(* Logix 5000 project; controller Lab05_anb5567_msw5288 vendor 1 type 14 code 77 rev 20.12; software revision 20.01 *)

TASK MainTask (continuous, watchdog 500 ms) : MainProgram

MODULES
   Controller : vendor 1 type 14 code 77 (CompactLogixL32EController 0, rev 20.12)
      LocalENB : 1769-L32E Ethernet Port (CompactLogixL32Ethernet 1, rev 20.11)
      Local : CompactBus (CompactVirtualAdapter 3, rev 20.11)
         DC_DI_16 : 1769-IQ16 (Compact 2, rev 1.1, Input RPI 20 ms)
         Analog_4I_2O : vendor 1 type 10 code 43 (Compact 1, rev 1.1, Output RPI 80 ms)
         Relay_DO_16 : 1769-OW16 (Compact 3, rev 1.1, Output RPI 20 ms)
         Analog_8Channel : 1769-IF8 (Compact 6, rev 1.1, Output RPI 80 ms)
         IT6C_TAI : vendor 1 type 10 code 36 (Compact 4, rev 1.1, Input RPI 80 ms)   // Thermocouple Input Module
END_MODULES

VAR_GLOBAL   (* controller tags *)
   ALM : DINT;   // Alarms
        .2   // P100 Run Fault
        .1   // Tank 100 high-high level alarm
        .0   // Low Low Level Alarm
   BV100 : BOOL;   // Tank 100 outlet valve(pneumatic solenoid)
   CV101 : BOOL;   // Tank 100 water inlet valve (pnematic solenoid)
   FCV101 : REAL;   // Tank 100 water in heater steam control valve (I/P)
   FT100 : REAL := -0.12483891;   // Tank 100 discharge flow rate (4-20 mA, 0 to 100 gpm)
   FT101 : REAL := -0.18725838;   // Tank 100 water in flow rate (4-20 mA, 0 to 150 gpm)
   gBit : DINT := 2;   // General Purpose Bits
        .2   // P100 IN AUTO
        .3   // Pump Transfer Started
        .4   // Stop (0 = stopped, 1 = OK)
        .5   // System Auto mode
        .0   // Start the Transfer
        .1   // Stop the Transfer
   gTmr : TIMER[10] := ([0].PRE := 3000, [1].PRE := 5000, [2].PRE := 3000, [3].PRE := 2000, [4].PRE := 500, [5].PRE := 500);   // Timers
        [1].DN   // Low Low Alarm Timer
   HMI_HOA_IA : DINT;   // In Auto
        .0   // Inlet Vave In Auto
        .1   // Outlet Valve In Auto
        .2   // Pump In Auto
   HMI_HOA_IH : DINT;   // In Hand
        .0   // Inlet Valve In Hand
        .1   // Outlet Valve In Hand
        .2   // Pump In Hand
   HMI_HOA_IO : DINT;   // In Off
        .0   // Inlet In Off
        .2   // Pump Off
        .1   // Outlet Valve In Off
   HMI_HOA_RA : DINT;   // Request Auto
        .0   // Request Inlet In Auto
        .1   // Request Outlet In Auto
        .2   // Request Pump In Auto
   HMI_HOA_RH : DINT;   // Request Hand
        .0   // Request Inlet In Hand
        .1   // Request Outlet In Hand
        .2   // Request Pump In hand
   HMI_HOA_RO : DINT;   // Request Off
        .0   // Request Inlet In Off
        .1   // Request Outlet OFF
        .2   // Request Pump Off
   HMI_MR : DINT := 2;   // Misc Request
        .0   // Request Transfer Start
        .1   // Request Transfer Stop
        .2   // Request System Auto
        .3   // Request Alarm Acknowledge
   HMI_MS : DINT := 2;   // Misc Status
        .0   // Start Transfer Status
        .1   // Stop Transfer Status
        .2   // System Auto Status
   HMI_PB : DINT;   // HMI Push Buttons
        .0   // CV101 Hand HMI PB
        .1   // CV101 OFF hmi PB
        .2   // CV101 Auto HMI PB
        .3   // BV100 Hand PB
        .4   // BV100 Off PB
        .5   // BV100 In Auto PB
        .6   // P100 Hand PB
        .7   // P100 OFF PB
        .8   // P100 Auto HMI PB
        .11   // Acknowledge
        .10   // Stop HMI Push Button
        .9   // Transfer HMI Push Button
   HOA_AC : DINT;   // Auto Command
        .0   // Inlet Auto Command
        .1   // Outlet Valve Auto Command
   LSH100 : BOOL;   // Tank 100 high level switch (1= water at switch)
   LSHH100 : BOOL := 1;   // Tank 100 high-high level switch (1= no water at switch)
   LSL100 : BOOL;   // Tank 100 low level switch (1 = water at switch)
   LSLL100 : BOOL := 1;   // Tank 100 low-low level switch (1 = water at switch)
   LT100 : REAL := 6.5884533;   // Tank 100 level (4-20 mA, 0 to 3 psi, 0 to 100% full at 6 ft.w.c.)
   N_ALM : DINT;   // New Alarms
        .2   // New P100 Run Fault
        .0   // New Low Low Level Alarm
        .1   // New Tank 100 high-high level alarm
   P100 : BOOL;   // Tank 100 outlet pump RUN (Motor starter coil)
   P100RNG : BOOL;   // Tank 100 Outlet pump RUNNING (motor starter auxiliary contact)
   PB100A : BOOL;   // Start PB (1 = pressed)
   PB100B : BOOL := 1;   // Stop PB (0 = pressed)
   PL100G : BOOL;   // Green Pilot light
   PL100R : BOOL;   // Red pilot light
   SimConfig : DINT[100];   // Simulation Configuration Data
        [1].0   // SIMULATION 1 = No 480 VAC to MCC
        [1].1   // SIMULATION 1 = Tank 100 disconnect is open
        [1].10   // SIMULATION 1 = LSLL100 switch bad
        [1].11   // SIMULATION 1 = LSL100 switch bad
        [1].12   // SIMULATION 1 = LSH100 switch bad
        [1].13   // SIMULATION 1 = LSHH100 switch bad
        [1].2   // SIMULATION 1 = Tank 100 fuses blown
        [1].3   // SIMULATION 1 = CV101 solenoid valve bad
        [1].4   // SIMULATION 1 = No plant air pressure for control valves
        [1].5   // SIMULATION 1 = BV100 solenoid valve bad
        [1].6   // SIMULATION 1 = Local:3:O 1769-OW16 output card fuse blown
        [1].7   // SIMULATION 1 = PL100G bulb bad
        [1].8   // SIMULATION 1 = PL100R bulb bad
        [1].9   // SIMULATION 1 = Local:2:I 1769-IQ16 +24 VDC to inputs fuse blown
   SimLocal_2_I_Data : INT := 1174;   // SIMULATED INPUTS 1769-IQ16 Local:2:I
        .0   // SIMULATED INPUT Local:2:I.Data.0 Start PB 1 = pressed PB100A
        .1   // SIMULATED INPUT Local:2:I.Data.1 Stop PB 0 = pressed PB100B
        .10   // SIMULATED INPUT Local:2:I.Data.10 Bin 100 outlet slide gate IS CLOSED
        .11   // SIMULATED INPUT Local:2:I.Data.11 Tank 100 agitator RUNNING
        .12   // SIMULATED INPUT Local:2:I.Data.12 spare
        .13   // SIMULATED INPUT Local:2:I.Data.13 spare
        .14   // SIMULATED INPUT Local:2:I.Data.14 spare
        .15   // SIMULATED INPUT Local:2:I.Data.15 spare
        .2   // SIMULATED INPUT Local:2:I.Data.2 Enable SS 1 = Enable SS100
        .3   // SIMULATED INPUT Local:2:I.Data.3 Tank 100 outlet pump RUNNING P100RNG
        .4   // SIMULATED INPUT Local:2:I.Data.4 Tank 100 low-low level switch 1=water at switch LSLL100
        .5   // SIMULATED INPUT Local:2:I.Data.5 Tank 100 low level switch 1=water at switch LSL100
        .6   // SIMULATED INPUT Local:2:I.Data.6 Tank 100 high level switch 1=water at switch LSH100
        .7   // SIMULATED INPUT Local:2:I.Data.7 Tank 100 high-high level switch 1=no water at switch LSHH100
        .8   // SIMULATED INPUT Local:2:I.Data.8 Bin 100 screw conveyor RUNNING
        .9   // SIMULATED INPUT Local:2:I.Data.9 Bin 100 outlet slide gate IS OPEN
   SPD100 : REAL;   // Tank 100 outlet pump speed command (VFD SPEED reference input)
   SS100 : BOOL := 1;   // Enable SS (1=enabled)
   TT100 : REAL := 57.889015;   // Tank 100 product temperature (4-20 mA, 0 to 250 °F)
   TT101 : REAL := 55.986225;   // Tank 100 water in temperature (4-20 mA, 0 to 250 °F)
   TT900 : REAL := 72.518555;   // Room temperature (Type T thermocouple)
   WT100 : REAL := 155.84729;   // Tank 100 weight (4-20 mA, 0 to 10000 lb)
END_VAR

PROGRAM MainProgram   (* main routine MainRoutine *)

ROUTINE AlarmLogic   (* ladder *)
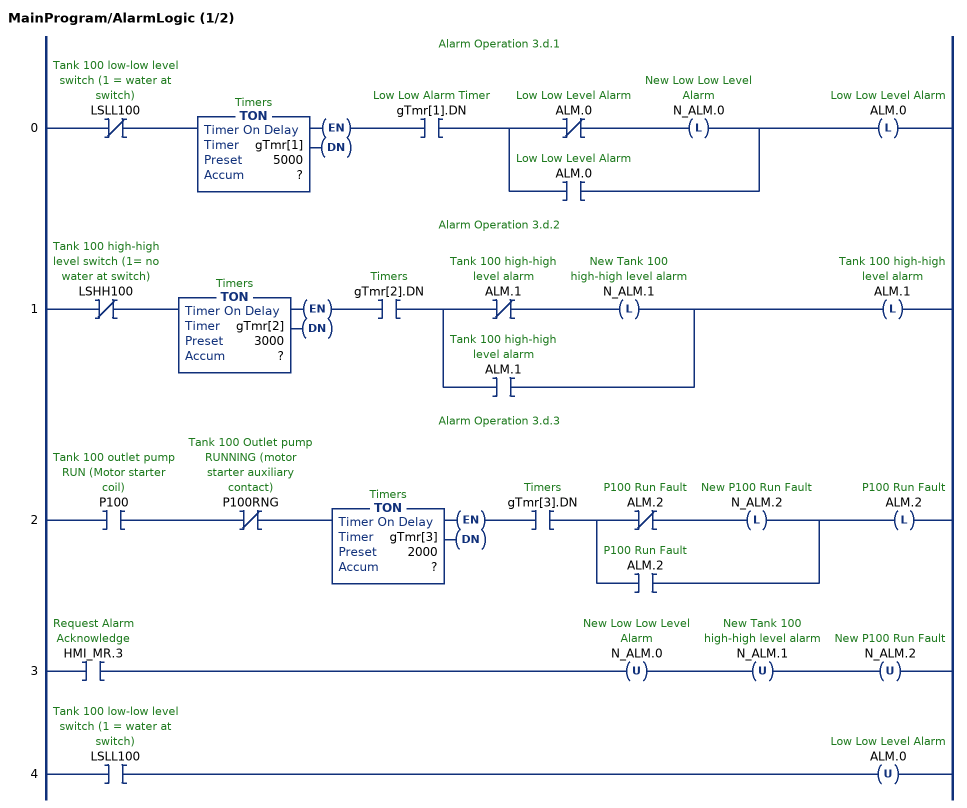
   // Alarm Operation 3.d.1
   0: XIO(LSLL100)TON(gTmr[1],?,?)XIC(gTmr[1].DN)[XIO(ALM.0) OTL(N_ALM.0) ,XIC(ALM.0) ]OTL(ALM.0);
   // Alarm Operation 3.d.2
   1: XIO(LSHH100)TON(gTmr[2],?,?)XIC(gTmr[2].DN)[XIO(ALM.1) OTL(N_ALM.1) ,XIC(ALM.1) ]OTL(ALM.1);
   // Alarm Operation 3.d.3
   2: XIC(P100)XIO(P100RNG)TON(gTmr[3],?,?)XIC(gTmr[3].DN)[XIO(ALM.2) OTL(N_ALM.2) ,XIC(ALM.2) ]OTL(ALM.2);
   3: XIC(HMI_MR.3)OTU(N_ALM.0)OTU(N_ALM.1)OTU(N_ALM.2);
   4: XIC(LSLL100)OTU(ALM.0);
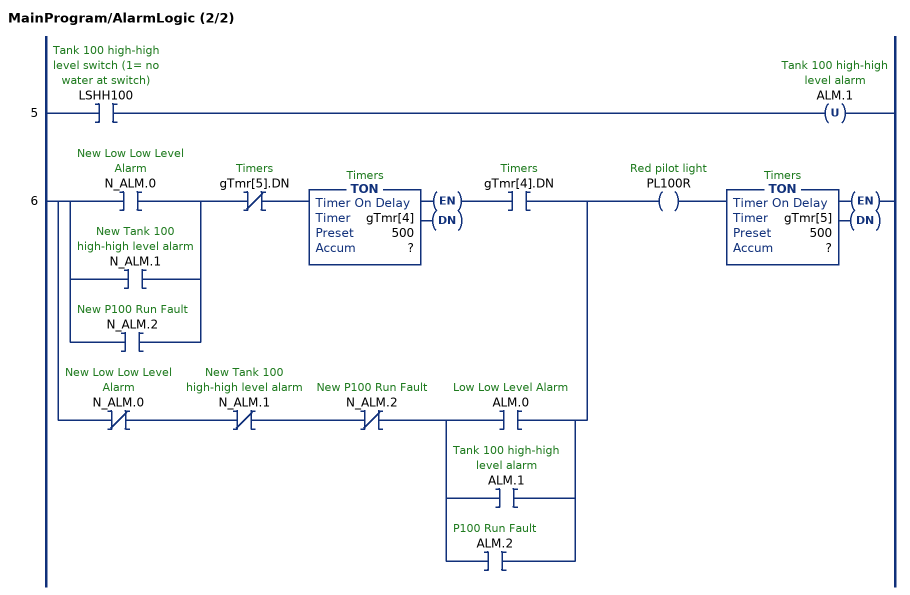
   5: XIC(LSHH100)OTU(ALM.1);
   6: [[XIC(N_ALM.0) ,XIC(N_ALM.1) ,XIC(N_ALM.2) ] XIO(gTmr[5].DN) TON(gTmr[4],?,?) XIC(gTmr[4].DN) ,XIO(N_ALM.0) XIO(N_ALM.1) XIO(N_ALM.2) [XIC(ALM.0) ,XIC(ALM.1) ,XIC(ALM.2) ] ]OTE(PL100R)TON(gTmr[5],?,?);
END_ROUTINE

ROUTINE HMIInputs   (* ladder *)
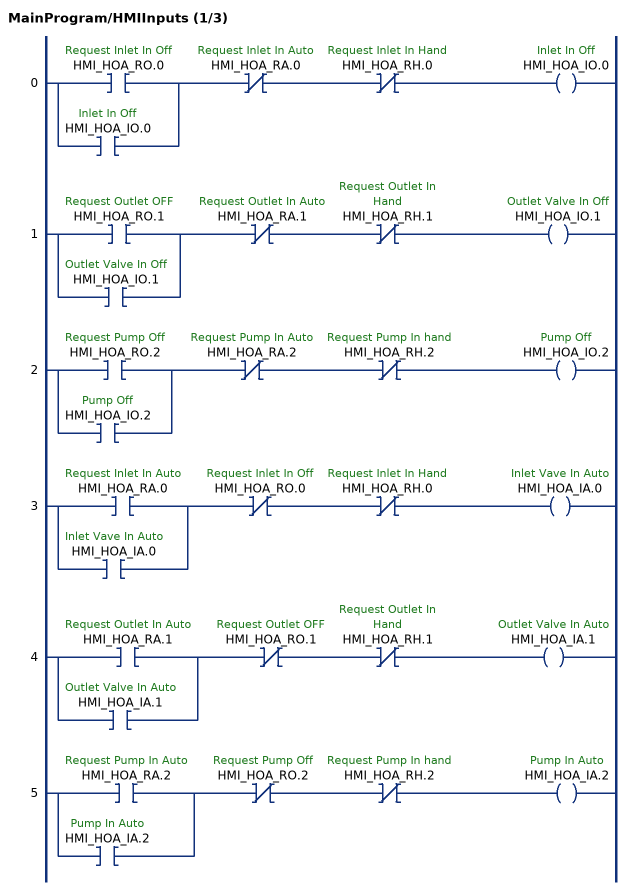
   0: [XIC(HMI_HOA_RO.0) ,XIC(HMI_HOA_IO.0) ]XIO(HMI_HOA_RA.0)XIO(HMI_HOA_RH.0)OTE(HMI_HOA_IO.0);
   1: [XIC(HMI_HOA_RO.1) ,XIC(HMI_HOA_IO.1) ]XIO(HMI_HOA_RA.1)XIO(HMI_HOA_RH.1)OTE(HMI_HOA_IO.1);
   2: [XIC(HMI_HOA_RO.2) ,XIC(HMI_HOA_IO.2) ]XIO(HMI_HOA_RA.2)XIO(HMI_HOA_RH.2)OTE(HMI_HOA_IO.2);
   3: [XIC(HMI_HOA_RA.0) ,XIC(HMI_HOA_IA.0) ]XIO(HMI_HOA_RO.0)XIO(HMI_HOA_RH.0)OTE(HMI_HOA_IA.0);
   4: [XIC(HMI_HOA_RA.1) ,XIC(HMI_HOA_IA.1) ]XIO(HMI_HOA_RO.1)XIO(HMI_HOA_RH.1)OTE(HMI_HOA_IA.1);
   5: [XIC(HMI_HOA_RA.2) ,XIC(HMI_HOA_IA.2) ]XIO(HMI_HOA_RO.2)XIO(HMI_HOA_RH.2)OTE(HMI_HOA_IA.2);
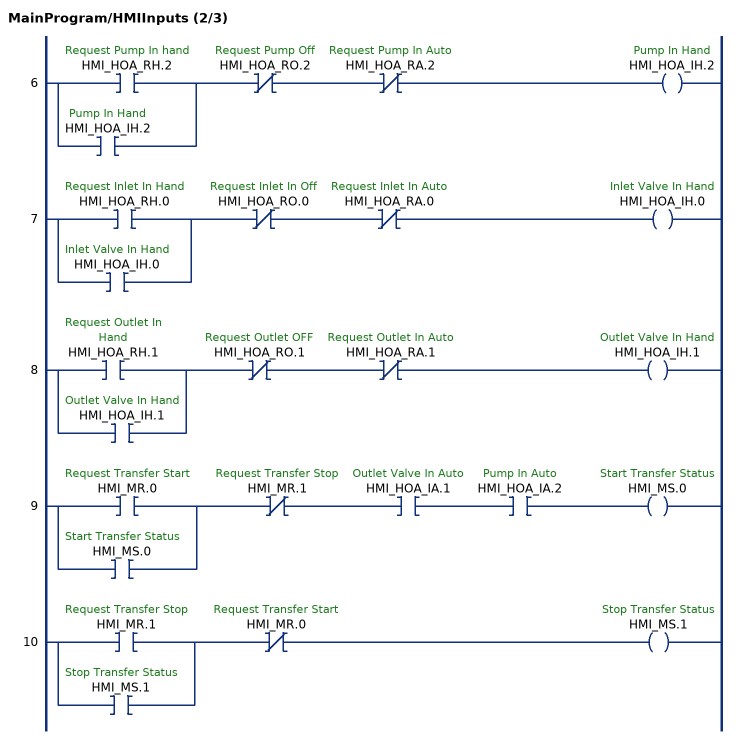
   6: [XIC(HMI_HOA_RH.2) ,XIC(HMI_HOA_IH.2) ]XIO(HMI_HOA_RO.2)XIO(HMI_HOA_RA.2)OTE(HMI_HOA_IH.2);
   7: [XIC(HMI_HOA_RH.0) ,XIC(HMI_HOA_IH.0) ]XIO(HMI_HOA_RO.0)XIO(HMI_HOA_RA.0)OTE(HMI_HOA_IH.0);
   8: [XIC(HMI_HOA_RH.1) ,XIC(HMI_HOA_IH.1) ]XIO(HMI_HOA_RO.1)XIO(HMI_HOA_RA.1)OTE(HMI_HOA_IH.1);
   9: [XIC(HMI_MR.0) ,XIC(HMI_MS.0) ]XIO(HMI_MR.1)XIC(HMI_HOA_IA.1)XIC(HMI_HOA_IA.2)OTE(HMI_MS.0);
   10: [XIC(HMI_MR.1) ,XIC(HMI_MS.1) ]XIO(HMI_MR.0)OTE(HMI_MS.1);
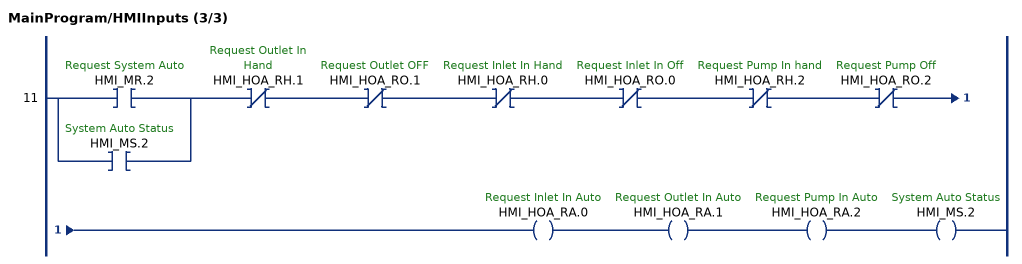
   11: [XIC(HMI_MR.2) ,XIC(HMI_MS.2) ]XIO(HMI_HOA_RH.1)XIO(HMI_HOA_RO.1)XIO(HMI_HOA_RH.0)XIO(HMI_HOA_RO.0)XIO(HMI_HOA_RH.2)XIO(HMI_HOA_RO.2)OTE(HMI_HOA_RA.0)OTE(HMI_HOA_RA.1)OTE(HMI_HOA_RA.2)OTE(HMI_MS.2);
END_ROUTINE

ROUTINE MainRoutine   (* ladder *)
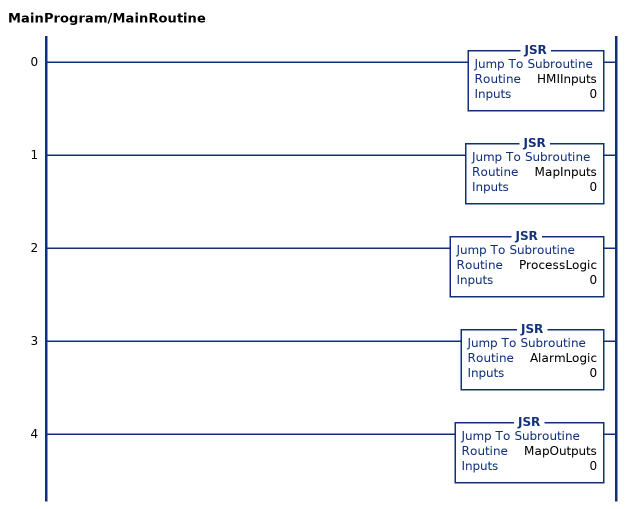
   0: JSR(HMIInputs,0);
   1: JSR(MapInputs,0);
   2: JSR(ProcessLogic,0);
   3: JSR(AlarmLogic,0);
   4: JSR(MapOutputs,0);
END_ROUTINE

ROUTINE MapInputs   (* ladder *)
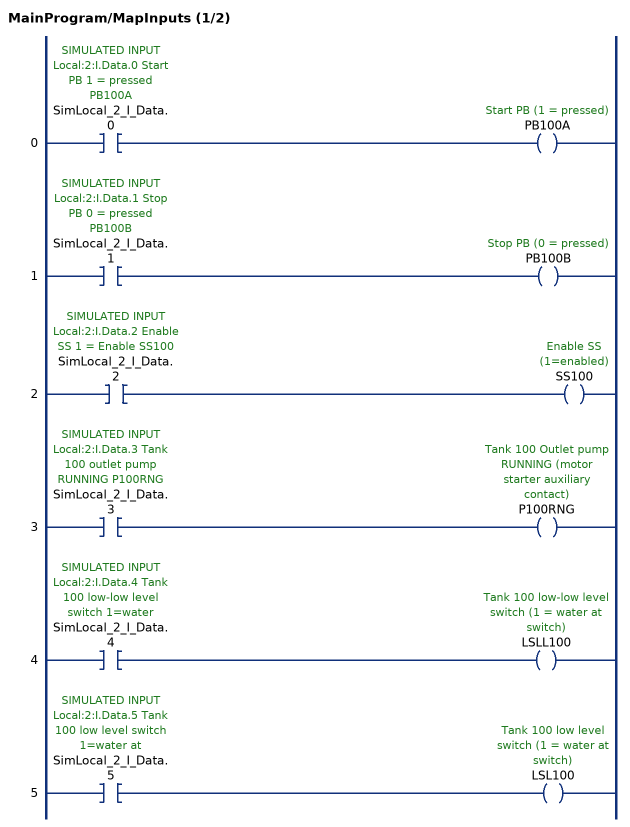
   0: XIC(SimLocal_2_I_Data.0)OTE(PB100A);
   1: XIC(SimLocal_2_I_Data.1)OTE(PB100B);
   2: XIC(SimLocal_2_I_Data.2)OTE(SS100);
   3: XIC(SimLocal_2_I_Data.3)OTE(P100RNG);
   4: XIC(SimLocal_2_I_Data.4)OTE(LSLL100);
   5: XIC(SimLocal_2_I_Data.5)OTE(LSL100);
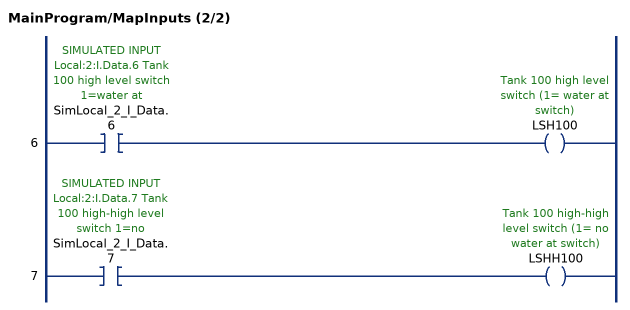
   6: XIC(SimLocal_2_I_Data.6)OTE(LSH100);
   7: XIC(SimLocal_2_I_Data.7)OTE(LSHH100);
END_ROUTINE

ROUTINE MapOutputs   (* ladder *)
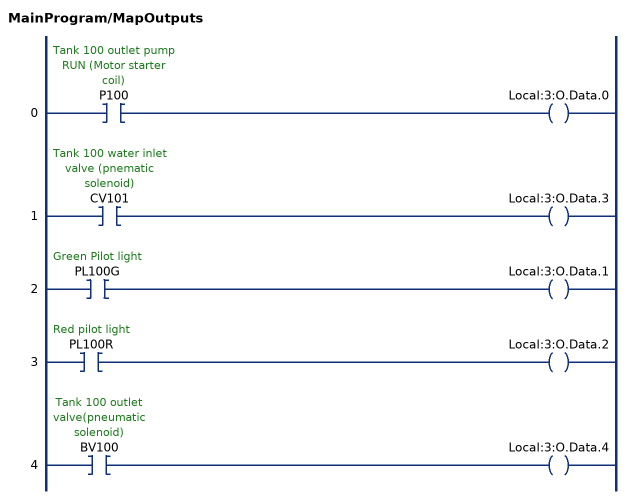
   0: XIC(P100)OTE(Local:3:O.Data.0);
   1: XIC(CV101)OTE(Local:3:O.Data.3);
   2: XIC(PL100G)OTE(Local:3:O.Data.1);
   3: XIC(PL100R)OTE(Local:3:O.Data.2);
   4: XIC(BV100)OTE(Local:3:O.Data.4);
END_ROUTINE

ROUTINE ProcessLogic   (* ladder *)
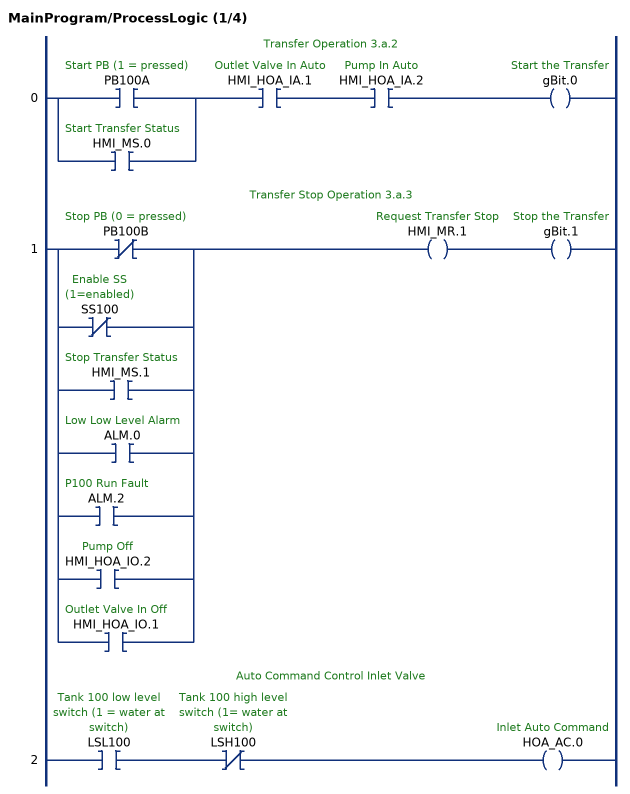
   // Transfer Operation 3.a.2
   0: [XIC(PB100A) ,XIC(HMI_MS.0) ]XIC(HMI_HOA_IA.1)XIC(HMI_HOA_IA.2)OTE(gBit.0);
   // Transfer Stop Operation 3.a.3
   1: [XIO(PB100B) ,XIO(SS100) ,XIC(HMI_MS.1) ,XIC(ALM.0) ,XIC(ALM.2) ,XIC(HMI_HOA_IO.2) ,XIC(HMI_HOA_IO.1) ]OTE(HMI_MR.1)OTE(gBit.1);
   // Auto Command Control Inlet Valve
   2: XIC(LSL100)XIO(LSH100)OTE(HOA_AC.0);
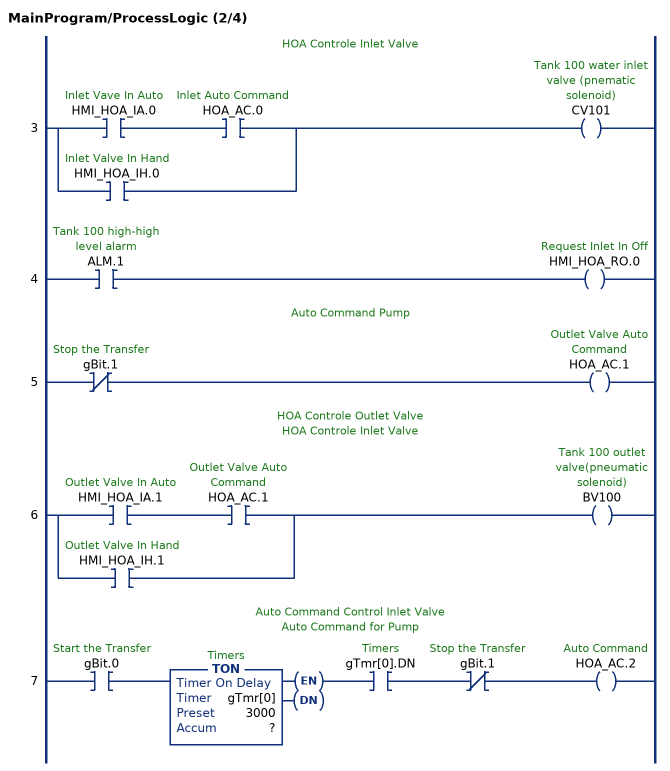
   // HOA Controle Inlet Valve
   3: [XIC(HMI_HOA_IA.0) XIC(HOA_AC.0) ,XIC(HMI_HOA_IH.0) ]OTE(CV101);
   4: XIC(ALM.1)OTE(HMI_HOA_RO.0);
   // Auto Command Pump
   5: XIO(gBit.1)OTE(HOA_AC.1);
   // HOA Controle Outlet Valve
   // HOA Controle Inlet Valve
   6: [XIC(HMI_HOA_IA.1) XIC(HOA_AC.1) ,XIC(HMI_HOA_IH.1) ]OTE(BV100);
   // Auto Command Control Inlet Valve
   // Auto Command for Pump
   7: XIC(gBit.0)TON(gTmr[0],?,?)XIC(gTmr[0].DN)XIO(gBit.1)OTE(HOA_AC.2);
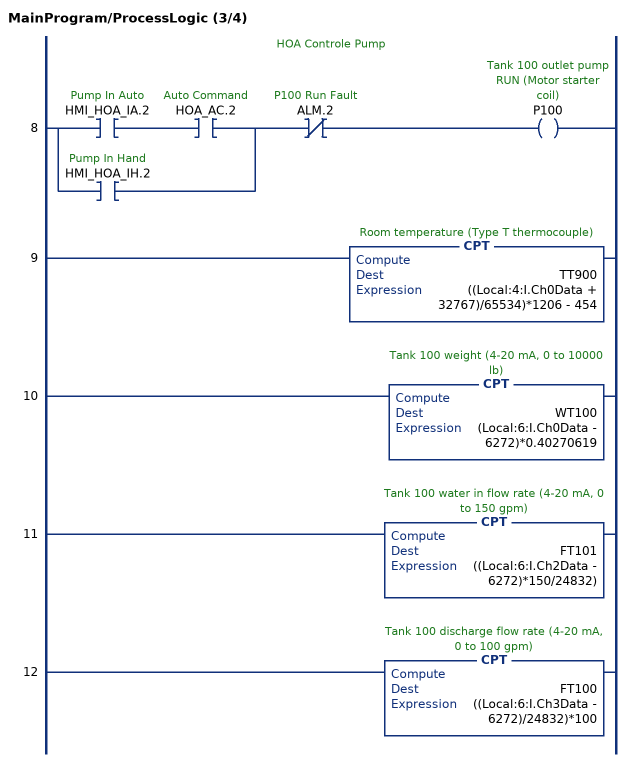
   // HOA Controle Pump
   8: [XIC(HMI_HOA_IA.2) XIC(HOA_AC.2) ,XIC(HMI_HOA_IH.2) ]XIO(ALM.2)OTE(P100);
   9: CPT(TT900,((Local:4:I.Ch0Data + 32767)/65534)*1206 - 454);
   10: CPT(WT100,(Local:6:I.Ch0Data - 6272)*0.40270619);
   11: CPT(FT101,((Local:6:I.Ch2Data - 6272)*150/24832));
   12: CPT(FT100,((Local:6:I.Ch3Data - 6272)/24832)*100);
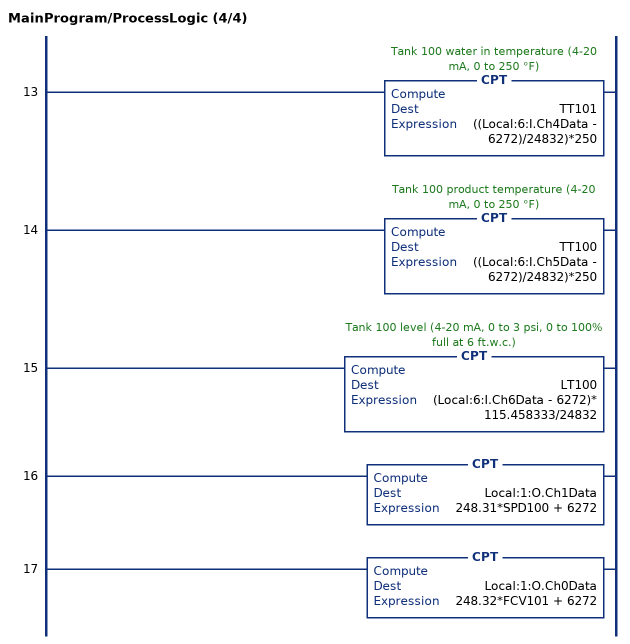
   13: CPT(TT101,((Local:6:I.Ch4Data - 6272)/24832)*250);
   14: CPT(TT100,((Local:6:I.Ch5Data - 6272)/24832)*250);
   15: CPT(LT100,(Local:6:I.Ch6Data - 6272)* 115.458333/24832);
   16: CPT(Local:1:O.Ch1Data,248.31*SPD100 + 6272);
   17: CPT(Local:1:O.Ch0Data,248.32*FCV101 + 6272);
END_ROUTINE
END_PROGRAM

PROGRAM Simulation   (* main routine Main *)
VAR
   simAGT100 : BOOL;   // SIMULATED DEVICE Tank 100 agitator RUN
   simAGT100RNG : BOOL;   // SIMULATED DEVICE Tank 100 agitator RUNNING
   simBit : DINT[20];   // General purpose simulation bits
        [0].0   // Reset scan min/max times
   simBV100 : BOOL;   // SIMULATED DEVICE Tank 100 outlet valve
   simBV102 : BOOL;   // SIMULATED DEVICE Tank 100 steam jacket block valve
   simCtr : COUNTER[100];   // General purpose simulation counters
   simCV101 : BOOL;   // SIMULATED DEVICE Tank 100 water inlet valve
   simCV103 : BOOL;   // SIMULATED DEVICE Tank 100 drain valve
   simCV110 : BOOL := 1;   // SIMULATED DEVICE Tank 100 to line 1 supply valve
   simCV120 : BOOL;   // SIMULATED DEVICE Tank 100 to line 2 supply valve
   simCV130 : BOOL;   // SIMULATED DEVICE Tank 100 to line 3 supply valve
   simCV140 : BOOL;   // SIMULATED DEVICE Tank 100 to line 4 supply valve
   simDint : DINT[100] := ([0] := 586517, [1] := 5, [2] := 16, [3] := 16, [4] := 44, [5] := 41, [6] := 34844, [7] := 34844, [8] := 956, [9] := 571, [10] := 971228);   // General purpose simulation 32-bit integers
        [0]   // Wall Clock Date/Time Year
        [10]   // Highest time since last scan (microSeconds)
        [1]   // Wall Clock Date/Time Month
        [2]   // Wall Clock Date/Time Day
        [3]   // Wall Clock Date/Time Hour
        [4]   // Wall Clock Date/Time Minute
        [5]   // Wall Clock Date/Time Second
        [6]   // Wall Clock Date/Time microSec
        [7]   // Wall Clock Date/Time microSec, last scan
        [8]   // Time since last scan (microSeconds)
        [9]   // Lowest time since last scan (microSeconds)
   simFCV101 : REAL;   // SIMULATED DEVICE Tank 100 water in steam control valve (% open)
   simFT100 : REAL;   // SIMULATED DEVICE Tank 100 discharge flow rate (gpm)
   simFT101 : REAL;   // SIMULATED DEVICE Tank 100 water in flow rate (gpm)
   simLSH100 : BOOL;   // SIMULATED DEVICE Tank 100 high level switch 1=water at switch
   simLSHH : BOOL := 1;   // SIMULATED DEVICE Tank 100 high-high level switch 1=no water at switch
   simLSL100 : BOOL;   // SIMULATED DEVICE Tank 100 low level switch 1=water at switch
   simLSLL100 : BOOL := 1;   // SIMULATED DEVICE Tank 100 low-low level switch 1=water at switch
   simLT100 : REAL := 0.17404613;   // SIMULATED DEVICE Tank 100 level (psi)
   simM101 : BOOL;   // SIMULATED DEVICE Bin 100 screw conveyor RUN
   simM101RNG : BOOL;   // SIMULATED DEVICE Bin 100 screw conveyor RUNNING
   simP100 : BOOL;   // SIMULATED DEVICE Tank 100 outlet pump RUN
   simP100RNG : BOOL;   // SIMULATED DEVICE Tank 100 outlet pump RUNNING
   simPB100A : BOOL;   // SIMULATED DEVICE Start PB 1=pressed
   simPB100B : BOOL := 1;   // SIMULATED DEVICE Stop PB 0=pressed
   simPL100G : BOOL;   // SIMULATED DEVICE Green pilot light
   simPL100R : BOOL;   // SIMULATED DEVICE Red pilot light
   simReal : REAL[100] := ([0] := 6.6983585, [1] := 20.095076, [7] := 0.999, [8] := 56.0, [9] := 0.9, [20] := 5.1999993, [21] := 4.4, [22] := 4.0000005, [23] := 4.0000005, [24] := 4.0000005, [25] := 4.0000005, [26] := 4.0000005, [27] := 4.0000005, [28] := 5.1999993, [29] := 5.1999993, [31] := 0.05, [32] := 0.22705016);   // General purpose simulation real numbers
        [0]   // SIMULATION Tank 100 Level, 0 to 100% full
        [10]   // SIMULATION of FT101 LPF x[n]
        [11]   // P100 SPEED command from user program
        [1]   // SIMULATION Gallons of water in tank 100
        [20]   // SIMULATION Screw conveyor 101 segment 0 (tank end) weight (lb)
        [21]   // SIMULATION Screw conveyor 101 segment 1 weight (lb)
        [22]   // SIMULATION Screw conveyor 101 segment 2 weight (lb)
        [23]   // SIMULATION Screw conveyor 101 segment 3 weight (lb)
        [24]   // SIMULATION Screw conveyor 101 segment 4 weight (lb)
        [25]   // SIMULATION Screw conveyor 101 segment 5 weight (lb)
        [26]   // SIMULATION Screw conveyor 101 segment 6 weight (lb)
        [27]   // SIMULATION Screw conveyor 101 segment 7 weight (lb)
        [28]   // SIMULATION Screw conveyor 101 segment 8 weight (lb)
        [29]   // SIMULATION Screw conveyor 101 segment 9 (bin end) weight (lb)
        [2]   // SIMULATION Pounds of dries in tank 100
        [30]   // SIMULATION Screw conveyor M101 speed (%)
        [31]   // SIMULATION (spare)
        [32]   // SIMULATION Screw conveyor 101 distance run since last data shift (ft)
        [33]   // SIMULATION Slide gate SG101 % open
        [3]   // SIMULATION (spare)
        [4]   // SIMULATION (spare)
        [5]   // SIMULATION (spare)
        [6]   // SIMULATION (spare)
        [7]   // SIMULATION of TT101 LPF alpha
        [8]   // SIMULATION of TT101 LPF x[n]
        [9]   // SIMULATION of FT100 LPF alpha
   simSG101 : BOOL;   // SIMULATED DEVICE Bin 100 outlet slide gate
   simSG101CL : BOOL := 1;   // SIMULATED DEVICE Bin 100 outlet slide gate IS CLOSED
   simSG101OP : BOOL;   // SIMULATED DEVICE Bin 100 outlet slide gate IS OPEN
   simSPD100 : REAL;   // SIMULATED DEVICE Tank 100 outlet pump speed command (% fs)
   simSS100 : BOOL := 1;   // SIMULATED DEVICE Enable SS 1=enabled
   simTmr : TIMER[100] := ([0].PRE := 50, [0].ACC := 35, [0].EN := 1, [0].TT := 1, [1].PRE := 500, [2].PRE := 1000, [3].PRE := 500, [3].ACC := 500, [3].EN := 1, [3].DN := 1, [4].PRE := 500, [5].PRE := 500, [6].PRE := 2000, [7].PRE := 2000, [7].ACC := 2000, [7].EN := 1, [7].DN := 1);   // General purpose simulation timers
        [0]   // Free running timer to update difference equations 0.05 sec pulse
        [1]   // P101RNG sim timer
        [2]   // simCV101 is open timer
        [3]   // simCV101 is closed timer
        [4]   // M101RNG sim timer
        [5]   // AGT100 sim timer
   simTT100 : REAL := 57.888206;   // SIMULATED DEVICE Tank 100 product temperature (deg F)
   simTT101 : REAL := 56.002384;   // SIMULATED DEVICE Tank 100 water in temperature (deg F)
   simWT100 : REAL := 167.59293;   // SIMULATED DEVICE Tank 100 weight (lb)
   simWT101 : REAL := 4500.0;   // SIMULATED DEVICE Bin 101 weight (lb)
END_VAR

ROUTINE FirstScanLogic   (* ladder *)
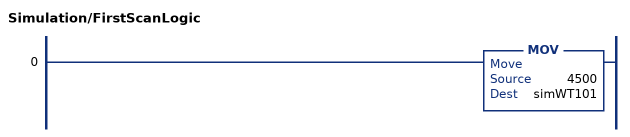
   0: MOV(4500,simWT101);
END_ROUTINE

ROUTINE Main   (* ladder *)
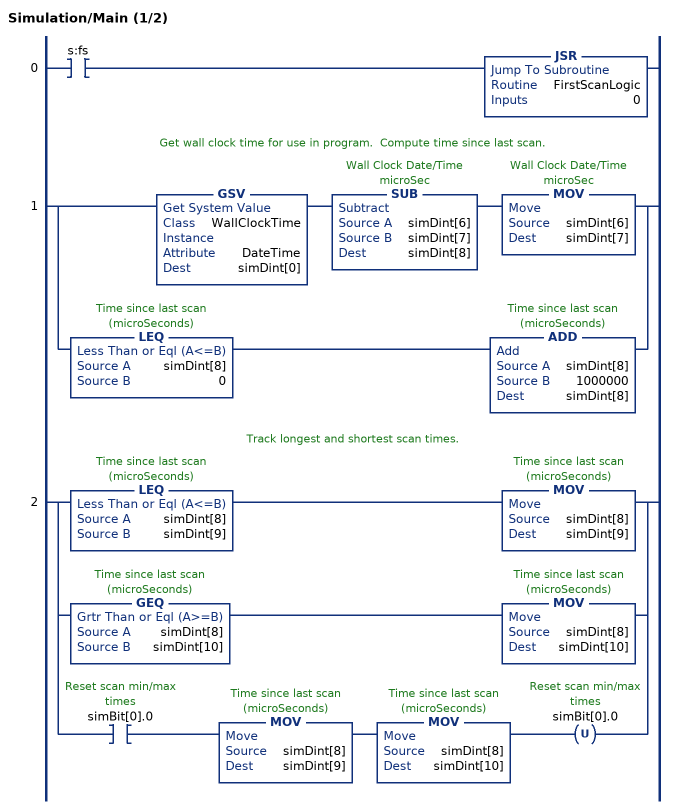
   0: XIC(s:fs)JSR(FirstScanLogic,0);
   // Get wall clock time for use in program.  Compute time since last scan.
   1: [GSV(WallClockTime,,DateTime,simDint[0]) SUB(simDint[6],simDint[7],simDint[8]) MOV(simDint[6],simDint[7]) ,LEQ(simDint[8],0) ADD(simDint[8],1000000,simDint[8]) ];
   // Track longest and shortest scan times.
   2: [LEQ(simDint[8],simDint[9]) MOV(simDint[8],simDint[9]) ,GEQ(simDint[8],simDint[10]) MOV(simDint[8],simDint[10]) ,XIC(simBit[0].0) MOV(simDint[8],simDint[9]) MOV(simDint[8],simDint[10]) OTU(simBit[0].0) ];
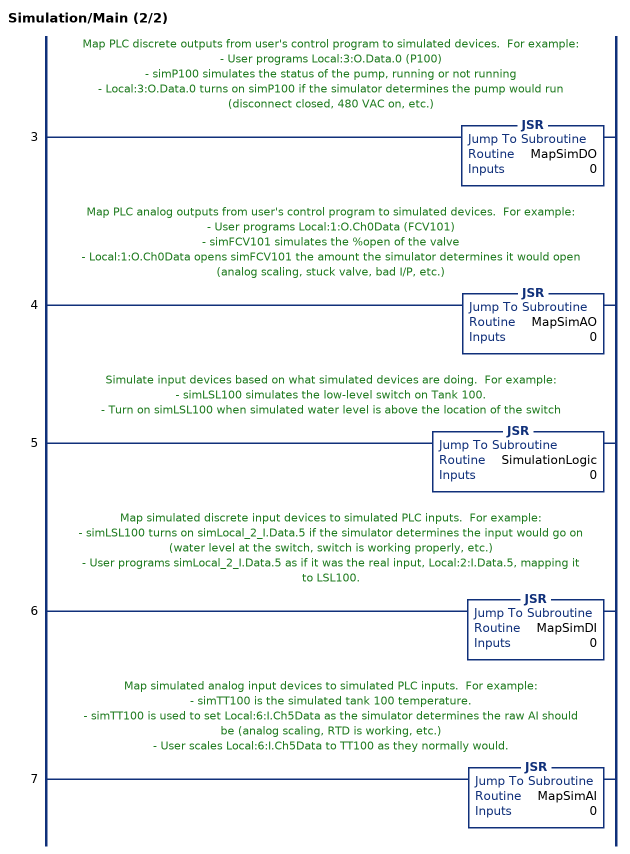
   // Map PLC discrete outputs from user's control program to simulated devices.  For example:
   //  - User programs Local:3:O.Data.0 (P100)
   //  - simP100 simulates the status of the pump, running or not running
   //  - Local:3:O.Data.0 turns on simP100 if the simulator determines the pump would run (disconnect closed, 480 VAC on, etc.)
   3: JSR(MapSimDO,0);
   // Map PLC analog outputs from user's control program to simulated devices.  For example:
   //  - User programs Local:1:O.Ch0Data (FCV101)
   //  - simFCV101 simulates the %open of the valve
   //  - Local:1:O.Ch0Data opens simFCV101 the amount the simulator determines it would open (analog scaling, stuck valve, bad I/P, etc.)
   4: JSR(MapSimAO,0);
   // Simulate input devices based on what simulated devices are doing.  For example:
   //  - simLSL100 simulates the low-level switch on Tank 100.
   //  - Turn on simLSL100 when simulated water level is above the location of the switch
   5: JSR(SimulationLogic,0);
   // Map simulated discrete input devices to simulated PLC inputs.  For example:
   //  - simLSL100 turns on simLocal_2_I.Data.5 if the simulator determines the input would go on (water level at the switch, switch is working properly, etc.)
   //  - User programs simLocal_2_I.Data.5 as if it was the real input, Local:2:I.Data.5, mapping it to LSL100.
   6: JSR(MapSimDI,0);
   // Map simulated analog input devices to simulated PLC inputs.  For example:
   //  - simTT100 is the simulated tank 100 temperature.
   //  - simTT100 is used to set Local:6:I.Ch5Data as the simulator determines the raw AI should be (analog scaling, RTD is working, etc.)
   //  - User scales Local:6:I.Ch5Data to TT100 as they normally would.
   7: JSR(MapSimAI,0);
END_ROUTINE

ROUTINE MapSimAI   (* ladder *)
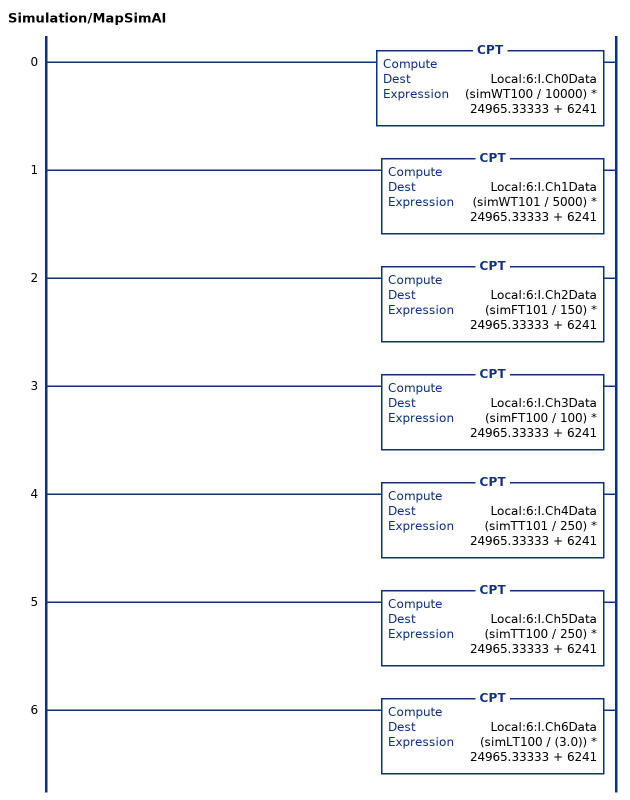
   0: CPT(Local:6:I.Ch0Data,(simWT100 / 10000) * 24965.33333 + 6241);
   1: CPT(Local:6:I.Ch1Data,(simWT101 / 5000) * 24965.33333 + 6241);
   2: CPT(Local:6:I.Ch2Data,(simFT101 / 150) * 24965.33333 + 6241);
   3: CPT(Local:6:I.Ch3Data,(simFT100 / 100) * 24965.33333 + 6241);
   4: CPT(Local:6:I.Ch4Data,(simTT101 / 250) * 24965.33333 + 6241);
   5: CPT(Local:6:I.Ch5Data,(simTT100 / 250) * 24965.33333 + 6241);
   6: CPT(Local:6:I.Ch6Data,(simLT100 / (3.0)) * 24965.33333 + 6241);
END_ROUTINE

ROUTINE MapSimAO   (* ladder *)
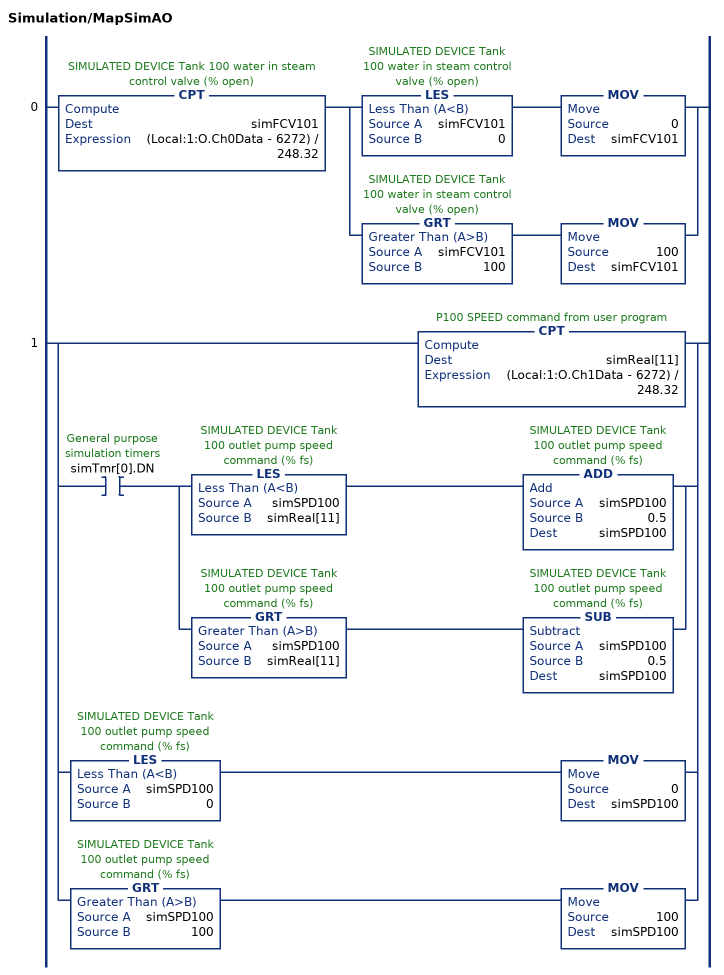
   0: CPT(simFCV101,(Local:1:O.Ch0Data - 6272) / 248.32)[LES(simFCV101,0) MOV(0,simFCV101) ,GRT(simFCV101,100) MOV(100,simFCV101) ];
   1: [CPT(simReal[11],(Local:1:O.Ch1Data - 6272) / 248.32) ,XIC(simTmr[0].DN) [LES(simSPD100,simReal[11]) ADD(simSPD100,0.5,simSPD100) ,GRT(simSPD100,simReal[11]) SUB(simSPD100,0.5,simSPD100) ] ,LES(simSPD100,0) MOV(0,simSPD100) ,GRT(simSPD100,100) MOV(100,simSPD100) ];
END_ROUTINE
